(* CODESYS project CFC_PROGRAMM.xml

Project tree, tasks and I/O mapping:
  program CFC_PROGRAMM [CFC]
*)

// CFC_PROGRAMM
PROGRAM CFC_PROGRAMM
VAR
	auxBool : BOOL;
	CLK : BOOL;
	R_TRIG_OUT : BOOL;
END_VAR
VAR_TEMP
	someBool : BOOL;
END_VAR
VAR // added by the converter: edge detectors and wires of the graphical bodies
    _w1, _w2 : ANY;
END_VAR

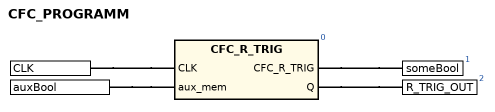
_w2 := CFC_R_TRIG(CLK := CLK, aux_mem := auxBool, Q => _w1);
someBool := _w2;
R_TRIG_OUT := _w1;

END_PROGRAM
